FUNCTION_BLOCK fbInheritanceLevel_4 EXTENDS fbInheritanceLevel_3
VAR
	{attribute addProperty Name "LEVEL 4"}
	level_4 : stAllTypes;
END_VAR

SUPER^();

METHOD Init : BOOL
VAR_INPUT
END_VAR
SUPER^.Init();
END_METHOD

END_FUNCTION_BLOCK

(* stored: Version 1.1.0.1, ProductVersion 3.1.4022.7
   POU fbInheritanceLevel_4: Id {ba63cbe9-92bb-4b9b-8666-6c548873f4d8}, SpecialFunc None
   Method Init: Id {b14964ff-8deb-4680-8a1b-107600890b21} *)
